{attribute addProperty BoxType "EK1122-0000-0018"}
{attribute addProperty Id "Beckhoff_EK12xxsub_EK1100EK1100_179A0949162"}
{attribute addProperty CRC "3919151873"}
{attribute addProperty SizeInBites "16"}
{attribute addProperty SizeInBytes "2"}
TYPE Beckhoff_EK12xxEK1122_E9998301 EXTENDS EK1122_179A0949 :
STRUCT
	{attribute addProperty Name "Beckhoff_EK12xxsub_EK1100"}
	Beckhoff_EK12xxsub_EK1100 : EK1100_179A0949;
END_STRUCT
END_TYPE

(* stored: Version 1.2.0.0, ProductVersion 3.1.4024.9
   DUT Beckhoff_EK12xxEK1122_E9998301: Id {55d9435b-9f68-4f66-a4a9-f4ceefb0cf50} *)
